// Block: Air_Data

DATA_BLOCK Air_Data
VERSION : 0.1
   NON_RETAIN
   VAR
      Air : Struct
         Pressure : Real;
         Flow : Real;
         TotalConsumption : LReal;
      END_STRUCT;
   END_VAR

BEGIN
   // No initialization required
END_DATA_BLOCK
